FUNCTION_BLOCK MockResettable IMPLEMENTS I_Resettable, I_Object
VAR
	_isRegistered : BOOL;
END_VAR

METHOD IsRegistered : BOOL
VAR_INPUT
END_VAR
IsRegistered := _isRegistered;
END_METHOD

METHOD RegisterWithParent
VAR_INPUT
	Parent	: I_HostObjects;
END_VAR
IF NOT _isRegistered THEN
	IF SUCCEEDED( Parent.RegisterResettable(THIS^)) THEN
		_isRegistered := TRUE;
	ELSE
		_isRegistered := FALSE;
	END_IF
END_IF
END_METHOD

METHOD Reset : Base_Library.HRESULT
END_METHOD

END_FUNCTION_BLOCK

(* stored: Version 1.1.0.1
   POU MockResettable: Id {67982418-1fe2-4e79-a8c0-e8754cff9aa1}, SpecialFunc None
   Method IsRegistered: Id {ff687a51-0cb0-434f-a789-f93048405b3c}
   Method RegisterWithParent: Id {deccf2f8-074a-48c7-b313-f7a823ef95ac}
   Method Reset: Id {1234c94a-2dee-47aa-a9a9-8e6b9ea31d76} *)
